Fanuc KAREL source: kf00102.KL

-- PROVISIONAL review KL for V940-1; original PC SHA256 cb1a14209d9bdec12890a1722fdb0df98f21685ec773c6bc31fcb83508d93e89
-- Incomplete behavior may be omitted. Consult companion uncertainty JSON. Do not deploy.
PROGRAM KF00102
%NOLOCKGROUP
BEGIN
  -- V9_ZERO_TABLE_METADATA_HINT layout=0002_ascii; no indexed target words; source/name/runtime held
  -- UNRESOLVED_PC offsets 5-16; opcodes 2E,23
  -- UNRESOLVED_PC offsets 21-32; opcodes 2E,23
  -- UNRESOLVED_PC offsets 37-63; opcodes 27,27,9D,22,1C,22,27,9D,31
  -- UNRESOLVED_PC offsets 68-72; opcodes 7F
END KF00102
